RoboDK station: Botellas_ICS.rdk

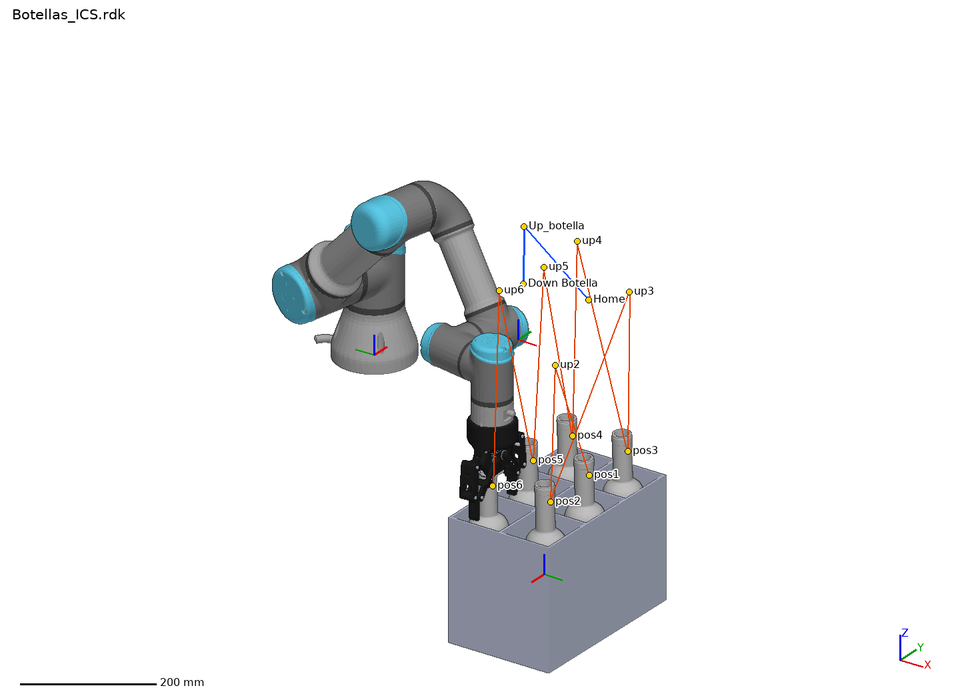
[picture v0: the station drawn from its stored meshes, robots at their saved joint values, targets as dots, program paths as lines]
Station Botellas_ICS (saved by RoboDK 5.5.1). Poses are relative to the parent item; angles as X-Y-Z fixed-axis rotations.
  - frame General_Frame at (0, 0, 0) mm
    - frame Basked_frame at (207.27, -229.59, -233.08) mm, rotated rx 0 ry 0 rz -90 deg
      - object basked at (110, 100, 0) mm, rotated rx 90 ry 0 rz 0 deg, size 299.8 x 204 x 180 mm, geometry from basked.STEP
      - target Home (Cartesian target) at (110.59, 156.63, 536.43) mm, rotated rx -179.23 ry -0.45 rz 2.88 deg; joints [64.989, -31.423, -16.963, -42.504, -90.042, -27.728] of UR3
      - target Up_botella (Cartesian target) at (-237.12, -202.06, 416.73) mm, rotated rx -179.95 ry -1.36 rz 80.65 deg; joints [18.228, -102.65, -36.587, -131.35, 88.777, 27.749] of UR3
      - target Down Botella (Cartesian target) at (-237.39, -203.22, 322.06) mm, rotated rx -179.95 ry -1.36 rz 80.65 deg; joints [18.422, -91.283, -78.287, -101.02, 88.779, 27.943] of UR3
      - target pos1 (Cartesian target) at (109.52, 157.88, 249.37) mm, rotated rx -179.23 ry -0.45 rz 2.88 deg; joints [-86.26, -143.334, -79.972, -45.934, 89.535, 1.021] of UR3
      - target pos2 (Cartesian target) at (209.72, 157.93, 246.4) mm, rotated rx -179.23 ry -0.45 rz 2.88 deg; joints [-99.075, -149.3, -67.668, -52.188, 89.715, -11.793] of UR3
      - target pos3 (Cartesian target) at (12.14, 158.01, 249.52) mm, rotated rx -179.23 ry -0.45 rz 2.88 deg; joints [-73.478, -142.07, -82.716, -44.575, 89.379, 13.802] of UR3
      - target pos4 (Cartesian target) at (13.74, 60.28, 248.5) mm, rotated rx -179.23 ry -0.45 rz 2.88 deg; joints [-68.857, -128.202, -116.575, -24.636, 89.329, 18.424] of UR3
      - target pos5 (Cartesian target) at (110.78, 57.98, 246.64) mm, rotated rx -179.23 ry -0.45 rz 2.88 deg; joints [-85.304, -129.535, -114.338, -25.374, 89.523, 1.977] of UR3
      - target pos6 (Cartesian target) at (213.89, 57.79, 245.54) mm, rotated rx -179.23 ry -0.45 rz 2.88 deg; joints [-102.13, -134.578, -102.169, -32.395, 89.761, -14.848] of UR3
      - target up2 (Cartesian target) at (199.82, 159.77, 466.29) mm, rotated rx -179.24 ry -0.46 rz 2.87 deg; joints [-97.825, -138.015, -19.35, -111.806, 89.691, -10.529] of UR3
      - target up3 (Cartesian target) at (13.93, 162.62, 512.11) mm, rotated rx -179.23 ry -0.45 rz 2.88 deg; joints [77.411, -33.585, -13.485, -43.79, -90.232, -15.307] of UR3
      - target up4 (Cartesian target) at (10.05, 66.19, 566.7) mm, rotated rx -179.22 ry -0.45 rz 2.9 deg; joints [-55.186, -100.538, -29.661, -139.381, 89.21, 32.081] of UR3
      - target up5 (Cartesian target) at (110.04, 76.19, 566.94) mm, rotated rx -179.23 ry -0.45 rz 2.88 deg; joints [-75.551, -102.496, -27.053, -139.791, 89.402, 11.729] of UR3
      - target up6 (Cartesian target) at (210.05, 66.2, 565.99) mm, rotated rx -179.23 ry -0.45 rz 2.88 deg; joints [42.966, -55.055, -15.775, -20.01, -89.705, -49.748] of UR3
      - object b6 at (446.84, 176.92, 34.82) mm, rotated rx 109.83 ry -88.86 rz -37.06 deg, size 246.5 x 62 x 63.4 mm, geometry from b.stl
      - object b5 at (547.04, 176.89, 31.86) mm, rotated rx 109.71 ry -88.87 rz -36.95 deg, size 246.5 x 62 x 63.4 mm, geometry from b.stl
      - object b1 at (349.41, 176.88, 34.88) mm, rotated rx 108.88 ry -88.86 rz -36.13 deg, size 246.5 x 62 x 63.4 mm, geometry from b.stl
      - object b4 at (351.01, 79.15, 33.87) mm, rotated rx 108.89 ry -88.86 rz -36.14 deg, size 246.5 x 62 x 63.4 mm, geometry from b.stl
      - object b2 at (448.05, 76.84, 32.01) mm, rotated rx 109.4 ry -88.85 rz -36.65 deg, size 246.5 x 62 x 63.4 mm, geometry from b.stl
      - object b3 at (551.16, 76.65, 30.91) mm, rotated rx 108.88 ry -88.86 rz -36.13 deg, size 246.5 x 62 x 63.4 mm, geometry from b.stl
  - frame UR3 Base at (-77.86, -257.16, 56.26) mm, rotated rx 0 ry 0 rz 90.17 deg
    - robot UR3: 6 axes, payload 3 kg, reach 500 mm, repeatability 0.1 mm, weight 11 kg
        modified DH rows (alpha deg, a mm, theta deg, d mm): 0, 0, 0, 151.9; 90, 0, 180, 0; 0, 243.65, 0, 0; 0, 213, 0, 110.4; -90, 0, 0, 83.4; 90, 0, 180, 82.4
        joint limits [-360, -360, -360, -360, -360, -360] to [360, 360, 360, 360, 360, 360]; home [0, -90, -90, 0, 90, 0]; saved at [-102.129, -134.578, -102.166, -32.401, 89.758, -14.841]
      - tool RobotiQ 2F-85 Gripper (Closed), TCP at (0, 0, 130) mm, size 134.4 x 157.6 x 75 mm
      - tool RobotiQ 2F-85 Gripper (Open), TCP at (0, 0, 110) mm, size 147.4 x 146.8 x 75 mm
  - program Re-ubicar (9 instructions, listed below)
  - program pick_place (9 instructions, listed below)
  - program soltar (3 instructions, listed below)
  - program proceso (26 instructions, listed below)
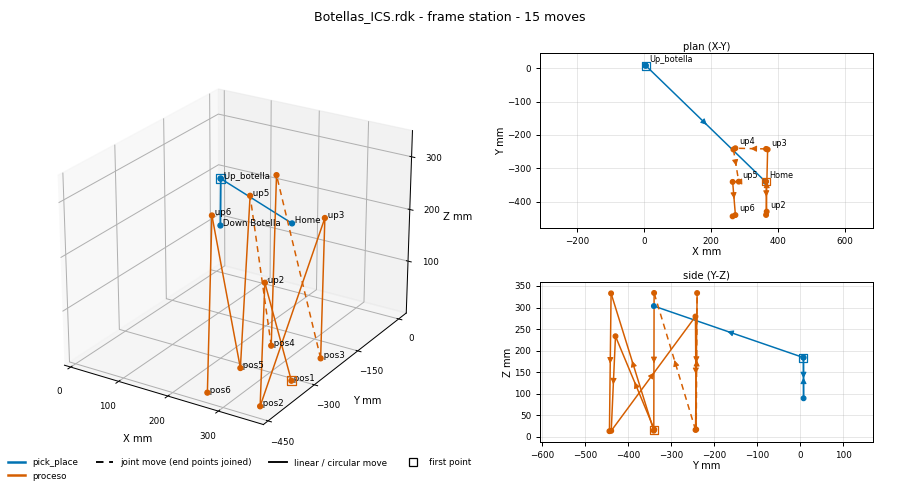
[picture p0: tool path of Botellas_ICS.rdk in frame station, 15 of 15 moves have a stored position in this frame; points joined in program order, loops and branches not executed]

--- program Re-ubicar (robot UR3) ---
  Reemplazar b1
  Reemplazar b4
  Reemplazar b2
  Reemplazar b3
  Reemplazar b5
  Reemplazar b6
  No definido
  Mostrar RobotiQ 2F-85 Gripper (Open)
  Ocultar RobotiQ 2F-85 Gripper (Closed)

--- program pick_place (robot UR3) ---
  Est. Ref.: Basked_frame
  Est. herr: RobotiQ 2F-85 Gripper (Open)
  MoveJ (Up_botella)
  MoveL (Down Botella)
  Mostrar RobotiQ 2F-85 Gripper (Closed)
  Ocultar RobotiQ 2F-85 Gripper (Open)
  Adjuntar a RobotiQ 2F-85 Gripper (Closed)
  MoveL (Up_botella)
  MoveL (Home)

--- program soltar (robot UR3) ---
  Separar de RobotiQ 2F-85 Gripper (Closed)
  Ocultar RobotiQ 2F-85 Gripper (Closed)
  Mostrar RobotiQ 2F-85 Gripper (Open)

--- program proceso (robot UR3) ---
  Est. Ref.: Basked_frame
  Est. herr: RobotiQ 2F-85 Gripper (Open)
  Llamar pick_place
  MoveL (pos1)
  Llamar soltar
  Llamar pick_place
  MoveL (Target 11) -> target up2
  MoveL (pos2)
  Llamar soltar
  Llamar pick_place
  MoveL (Target 11) -> target up3
  MoveL (pos3)
  Llamar soltar
  Llamar pick_place
  MoveJ (Target 12) -> target up4
  MoveL (pos4)
  Llamar soltar
  Llamar pick_place
  MoveJ (Target 13) -> target up5
  MoveL (pos5)
  Llamar soltar
  Llamar pick_place
  MoveL (up6)
  MoveL (pos6)
  Llamar soltar
  Llamar Program1
